Staubli VAL3: dateBase.dtx

public bool bCenterPoint = true
public bool bFrameTeach = true
public bool bPLC
public bool bToolTeach
public bool bWorTbMoving
public frame fWorkTable = {x=1612.647528, y=43.391654, z=-98.162922, rx=0.062117, ry=-0.932889, rz=-75.762654, fatherId=world[0]}
public jointRx jHome = {j1=40.634813, j2=24.616005, j3=104.715218, j4=-108.663007, j5=68.526435, j6=132.709111}
public mdesc mGrindingSpd = {accel=80, decel=70, tmax=100, leave=0.5, reach=0.5}
public mdesc mNomSpeed = {accel=36, vel=60, decel=36, rmax=2000, tmax=100, blend=cartesian, leave=5, reach=5}
public num nPrdRadius = 299.265855
public tool tTCP = {x=-12.113679, y=2.514779, z=192.872851, rx=33.798326, ry=31.269905, rz=-56.042932, fatherId=flange[0], ioLink=valve1}
